(*
  Hardware mapping definition.
*)
TYPE ST_MappingDefinition :
STRUCT
  // absolute hw mapping
  nPhInst : UDINT := 1;      // ph hw instance selection
  nPcInst : UDINT := 1;      // pc hw instance selection
  // module internal mapping (relative to given nPm)
  nPm     : UDINT := 1;      // to pm x
  nPg     : UDINT := 1;      // to pg in pm x
  nPa     : UDINT := 1;      // to pa in pg
  nPs     : UDINT := 1;      // to ps in pa
  nPc     : UDINT := 1;      // to pc in pm
  nPcCh   : UDINT := 1;      // to pc channel of pc 1-4
END_STRUCT
END_TYPE

(* stored: Version 1.1.0.1, ProductVersion 3.1.4024.11
   DUT ST_MappingDefinition: Id {58270ba5-480a-4769-ab5b-8c33e70e36ca} *)
